PROGRAM PRG_Commands
VAR
	fbTofStartCommand1		: TOF;		// Shows the exection was happen
END_VAR

Commands.fbStartCommand1.Call();
	
fbTofStartCommand1(
	IN := Commands.fbStartCommand1.Q,
	PT := T#1S);	
	
Commands.fbCustomStateCommand1.Call();	
Commands.fbAddCommand1.Call();
Commands.fbDelayedAddCommand1.Call();

END_PROGRAM

(* stored: Version 1.1.0.1, ProductVersion 3.1.4022.10
   POU PRG_Commands: Id {411fcb37-780f-06ea-2006-e35ff122d5e1}, SpecialFunc None *)
